(* Logix 5000 project; controller DC01 vendor 1 type 14 code 165 rev 32.12; software revision 32.04; part 12 of 13 *)
(* tags used below, declared in another part *)
   Always_Off : BOOL;
   Break_1stStation : BOOL;
   Break_LineWide : BOOL;
   Break_WorkCenter : BOOL;
   Break_Workstation : BOOL;
   FaultExists : CONTROL;
   LN04_MainLine_MSG : MESSAGE;
   Local_Timer : TIMER[30];
   ONS_0 : DINT;
   Scheduled_Units_Buffer : DINT;
   Shift_Reset : BOOL;
   Shift_Reset_ONS : BOOL;
   LN04_1st_Station_Break_Code : DINT;
   LN04_Additional_Break_Limit_Mins : DINT;
   LN04_BakeDrawer_MNT : DINT;
   LN04_Boxing_MNT : DINT;
   LN04_Console_MNT : DINT;
   LN04_Cooktop_MNT : DINT;
   LN04_Current_Shift_Duration_Mins : DINT;
   LN04_Current_Shift_Duration_wBreaks_Mins : DINT;
   LN04_DC_Controlled_Theoretical_Units : BOOL;
   LN04_Door_MNT : DINT;
   LN04_EStop_Funct_Test : DINT;
   LN04_EStop_Main_Panel : DINT;
   LN04_EStop_Main_Safety_Relay : DINT;
   LN04_EStop_MCC_Cabinet : DINT;
   LN04_FrontFrame_MNT : DINT;
   LN04_FunctionalTest_MNT : DINT;
   LN04_Ignition_NewSNModel : BOOL[32];
   LN04_Ignition_SNModelMSG : STRING[5];
   LN04_MachineOverAll_MNT : DINT;
   LN04_Main_Messages : DINT[250];
   LN04_MainBack_MNT : DINT;
   LN04_Messages_Barcode_SNModel : Barcode_SNModel;
   LN04_OT_Shift_Break_In_Minutes : DINT;
   LN04_OvenCavity_MNT : DINT;
   LN04_Pull_Cord_EStop_9111 : DINT;
   LN04_Pull_Cord_EStop_9112 : DINT;
   LN04_Pull_Cord_EStop_9200 : DINT;
   LN04_Pull_Cord_EStop_9201 : DINT;
   LN04_RackAndLiterature_MNT : DINT;
   LN04_Schedule : UDT_Current_Status;
   LN04_Schedule_Cycle_Timer : TIMER;
   LN04_Schedule_Max_Break_Duration : DINT;
   LN04_Schedule_Max_Break_Timer : TIMER;
   LN04_Schedule_TAKT : REAL;
   LN04_SidePanel_MNT : DINT;
   LN04_Standard_Shift_Break_In_Minutes : DINT;
   LN04_StorageDrawer_MNT : DINT;
   LN04_Theoretical_Units_Counter : COUNTER;
   LN04_Theoretical_Units_Counter_ONS : BOOL;
   LN04_Units_for_repair : DINT;
   LN04_Wiring_MNT : DINT;
   LN04EAM01 : DINT;
   LN04EAM02 : DINT;
   LN04ECM01 : DINT;
   LN04ECM02 : DINT;
   LN04EDM01 : DINT;
   LN04EEM01 : DINT;
   LN04EEM02 : DINT;
   LN04EEM03 : DINT;
   LN04EFM03 : DINT;
   LN04EGM01 : DINT;
   LN04EGM04 : DINT;
   LN04EGS01 : DINT;
   LN04EGS02 : DINT;
   LN04EGS03 : DINT;
   LN04EHM01 : DINT;
   LN04EHM02 : DINT;
   LN04EHM03 : DINT;
   LN04EHM04 : DINT;
   LN04EMM01 : DINT;
   LN04EMM03 : DINT;
   LN04NBS01 : DINT;
   LN04NBS02 : DINT;
   LN04NNM02 : DINT;
   LN04SAS01 : DINT;
   LN04SAS02 : DINT;
   LN04SDS01 : DINT;
   LN04SLS01 : DINT;
   LN04SLS02 : DINT;
   LN04SLS03 : DINT;
   LN04SNM02 : DINT;
   LN04WAM01 : DINT;
   LN04WBM01 : DINT;
   LN04WBM02 : DINT;
   LN04WCS01 : DINT;
   LN04WEM01 : DINT;
   LN04WEM02 : DINT;
   LN04WEM03 : DINT;
   LN04WFM01 : DINT;
   LN04WFM02 : DINT;
   LN04WFM03 : DINT;
   LN04WFM04 : DINT;
   LN04WFM05 : DINT;
   LN04WFS01 : DINT;
   LN04WFS02 : DINT;
   LN04WJM01 : DINT;
   LN04WJM02 : DINT;
   LN04WJM03 : DINT;
   LN04WKM01 : DINT;
   LN04WKM02 : DINT;
   LN04WKM03 : DINT;
   LN04WLM01 : DINT;
   LN04WMM01 : DINT;
   LN04WMM02 : DINT;
   LN04WMM03 : DINT;
   LN04WMM04 : DINT;
   LN04WNM01 : DINT;
(* LN04, continued *)

ROUTINE R02_CurrentShift_Calcs   (* ladder *)
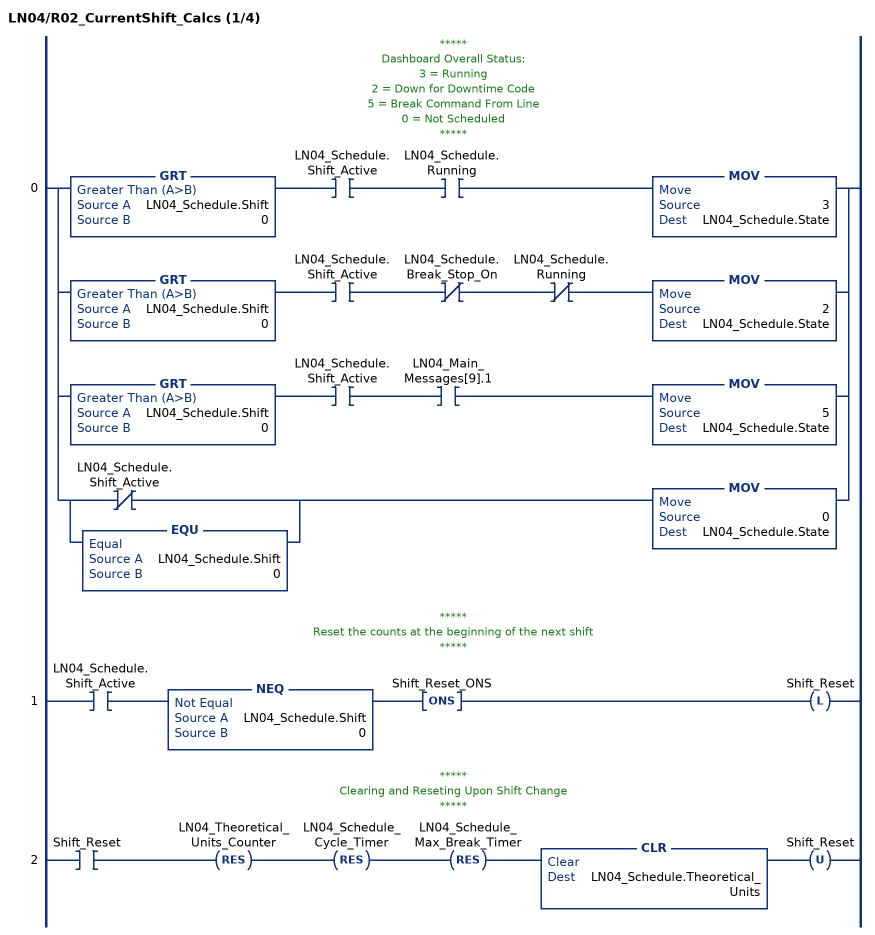
   // *****
   // Dashboard Overall Status:
   // 3 = Running
   // 2 = Down for Downtime Code
   // 5 = Break Command From Line
   // 0 = Not Scheduled
   // *****
   0: [GRT(LN04_Schedule.Shift,0) XIC(LN04_Schedule.Shift_Active) XIC(LN04_Schedule.Running) MOV(3,LN04_Schedule.State) ,GRT(LN04_Schedule.Shift,0) XIC(LN04_Schedule.Shift_Active) XIO(LN04_Schedule.Break_Stop_On) XIO(LN04_Schedule.Running) MOV(2,LN04_Schedule.State) ,GRT(LN04_Schedule.Shift,0) XIC(LN04_Schedule.Shift_Active) XIC(LN04_Main_Messages[9].1) MOV(5,LN04_Schedule.State) ,[XIO(LN04_Schedule.Shift_Active) ,EQU(LN04_Schedule.Shift,0) ] MOV(0,LN04_Schedule.State) ];
   // *****
   // Reset the counts at the beginning of the next shift
   // *****
   1: XIC(LN04_Schedule.Shift_Active)NEQ(LN04_Schedule.Shift,0)ONS(Shift_Reset_ONS)OTL(Shift_Reset);
   // *****
   // Clearing and Reseting Upon Shift Change
   // *****
   2: XIC(Shift_Reset)RES(LN04_Theoretical_Units_Counter)RES(LN04_Schedule_Cycle_Timer)RES(LN04_Schedule_Max_Break_Timer)CLR(LN04_Schedule.Theoretical_Units)OTU(Shift_Reset);
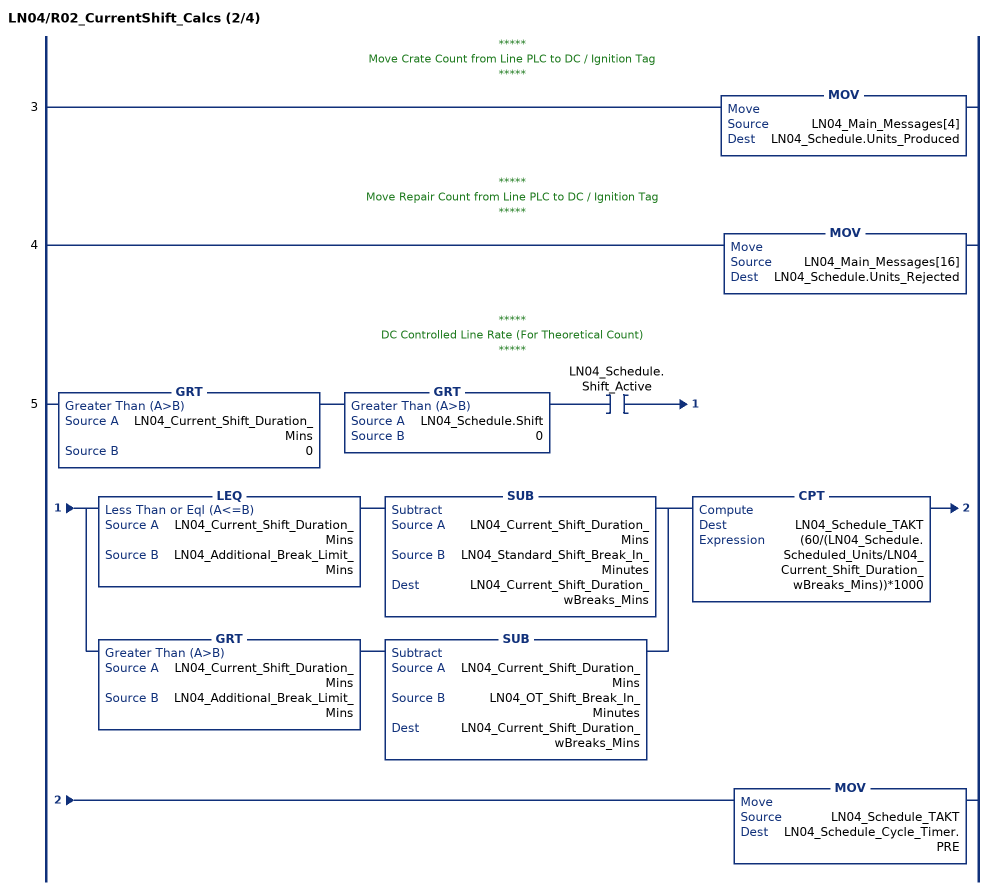
   // *****
   // Move Crate Count from Line PLC to DC / Ignition Tag
   // *****
   3: MOV(LN04_Main_Messages[4],LN04_Schedule.Units_Produced);
   // *****
   // Move Repair Count from Line PLC to DC / Ignition Tag
   // *****
   4: MOV(LN04_Main_Messages[16],LN04_Schedule.Units_Rejected);
   // *****
   // DC Controlled Line Rate (For Theoretical Count)
   // *****
   5: GRT(LN04_Current_Shift_Duration_Mins,0)GRT(LN04_Schedule.Shift,0)XIC(LN04_Schedule.Shift_Active)[LEQ(LN04_Current_Shift_Duration_Mins,LN04_Additional_Break_Limit_Mins) SUB(LN04_Current_Shift_Duration_Mins,LN04_Standard_Shift_Break_In_Minutes,LN04_Current_Shift_Duration_wBreaks_Mins) ,GRT(LN04_Current_Shift_Duration_Mins,LN04_Additional_Break_Limit_Mins) SUB(LN04_Current_Shift_Duration_Mins,LN04_OT_Shift_Break_In_Minutes,LN04_Current_Shift_Duration_wBreaks_Mins) ]CPT(LN04_Schedule_TAKT,(60/(LN04_Schedule.Scheduled_Units/LN04_Current_Shift_Duration_wBreaks_Mins))*1000)MOV(LN04_Schedule_TAKT,LN04_Schedule_Cycle_Timer.PRE);
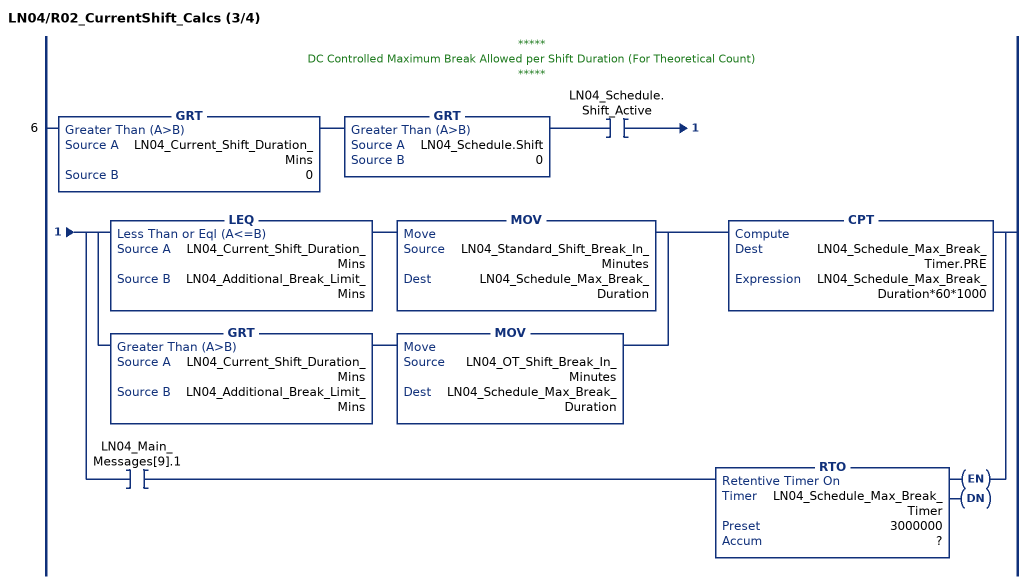
   // *****
   // DC Controlled Maximum Break Allowed per Shift Duration (For Theoretical Count)
   // *****
   6: GRT(LN04_Current_Shift_Duration_Mins,0)GRT(LN04_Schedule.Shift,0)XIC(LN04_Schedule.Shift_Active)[[LEQ(LN04_Current_Shift_Duration_Mins,LN04_Additional_Break_Limit_Mins) MOV(LN04_Standard_Shift_Break_In_Minutes,LN04_Schedule_Max_Break_Duration) ,GRT(LN04_Current_Shift_Duration_Mins,LN04_Additional_Break_Limit_Mins) MOV(LN04_OT_Shift_Break_In_Minutes,LN04_Schedule_Max_Break_Duration) ] CPT(LN04_Schedule_Max_Break_Timer.PRE,LN04_Schedule_Max_Break_Duration*60*1000) ,XIC(LN04_Main_Messages[9].1) RTO(LN04_Schedule_Max_Break_Timer,?,?) ];
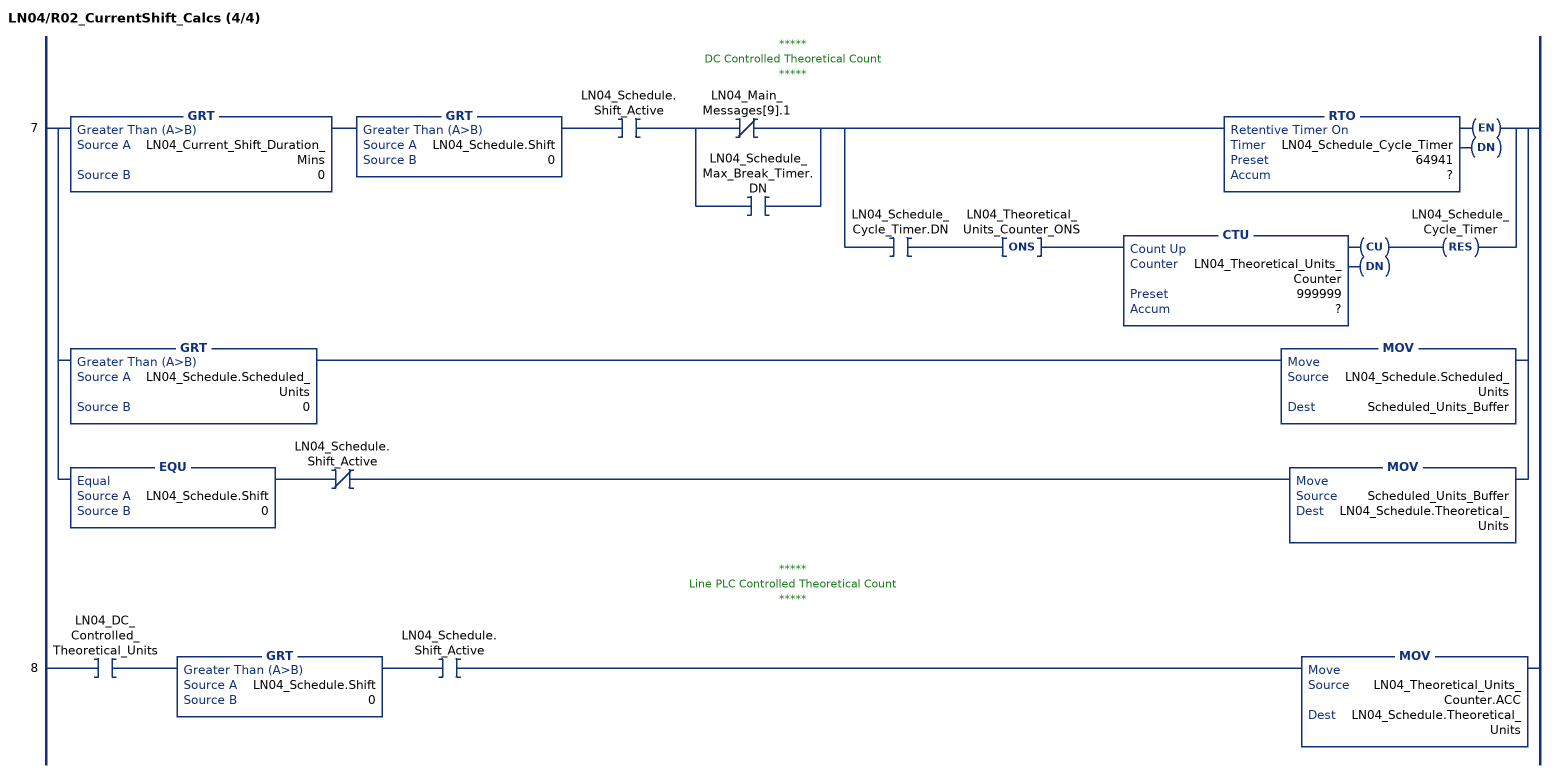
   // *****
   // DC Controlled Theoretical Count
   // *****
   7: [GRT(LN04_Current_Shift_Duration_Mins,0) GRT(LN04_Schedule.Shift,0) XIC(LN04_Schedule.Shift_Active) [XIO(LN04_Main_Messages[9].1) ,XIC(LN04_Schedule_Max_Break_Timer.DN) ] [RTO(LN04_Schedule_Cycle_Timer,?,?) ,XIC(LN04_Schedule_Cycle_Timer.DN) ONS(LN04_Theoretical_Units_Counter_ONS) CTU(LN04_Theoretical_Units_Counter,?,?) RES(LN04_Schedule_Cycle_Timer) ] ,GRT(LN04_Schedule.Scheduled_Units,0) MOV(LN04_Schedule.Scheduled_Units,Scheduled_Units_Buffer) ,EQU(LN04_Schedule.Shift,0) XIO(LN04_Schedule.Shift_Active) MOV(Scheduled_Units_Buffer,LN04_Schedule.Theoretical_Units) ];
   // *****
   // Line PLC Controlled Theoretical Count
   // *****
   8: XIC(LN04_DC_Controlled_Theoretical_Units)GRT(LN04_Schedule.Shift,0)XIC(LN04_Schedule.Shift_Active)MOV(LN04_Theoretical_Units_Counter.ACC,LN04_Schedule.Theoretical_Units);
END_ROUTINE

ROUTINE R03_DataFromLines   (* ladder *)
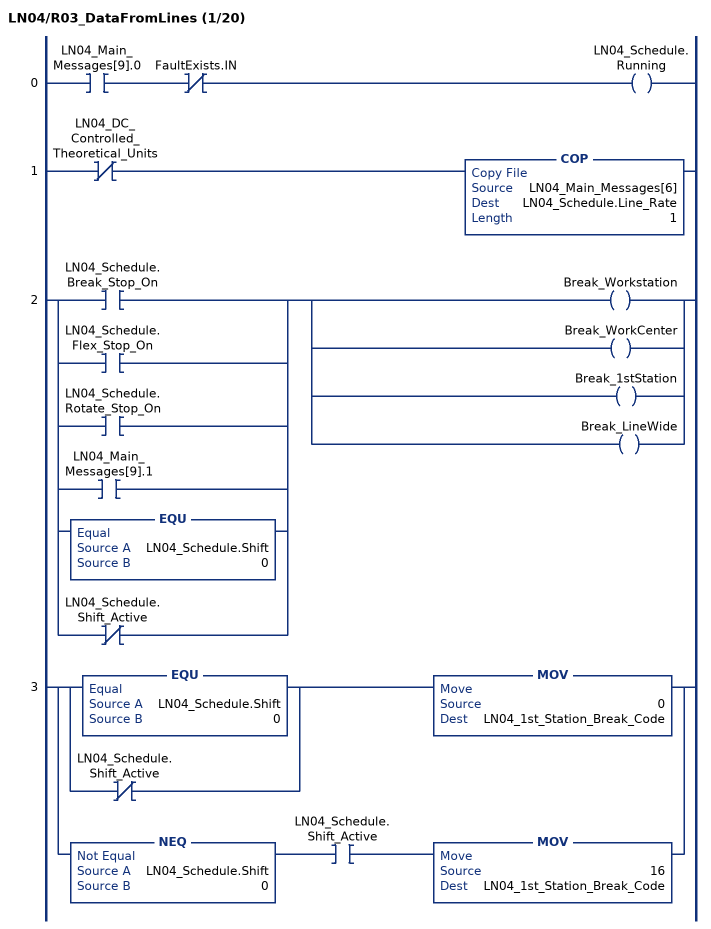
   0: XIC(LN04_Main_Messages[9].0)XIO(FaultExists.IN)OTE(LN04_Schedule.Running);
   1: XIO(LN04_DC_Controlled_Theoretical_Units)COP(LN04_Main_Messages[6],LN04_Schedule.Line_Rate,1);
   2: [XIC(LN04_Schedule.Break_Stop_On) ,XIC(LN04_Schedule.Flex_Stop_On) ,XIC(LN04_Schedule.Rotate_Stop_On) ,XIC(LN04_Main_Messages[9].1) ,EQU(LN04_Schedule.Shift,0) ,XIO(LN04_Schedule.Shift_Active) ][OTE(Break_Workstation) ,OTE(Break_WorkCenter) ,OTE(Break_1stStation) ,OTE(Break_LineWide) ];
   3: [[EQU(LN04_Schedule.Shift,0) ,XIO(LN04_Schedule.Shift_Active) ] MOV(0,LN04_1st_Station_Break_Code) ,NEQ(LN04_Schedule.Shift,0) XIC(LN04_Schedule.Shift_Active) MOV(16,LN04_1st_Station_Break_Code) ];
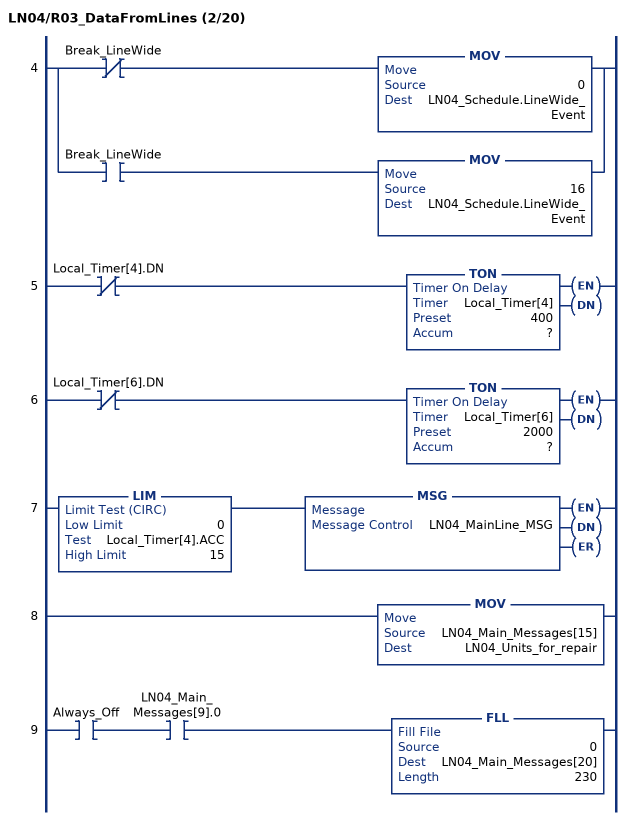
   4: [XIO(Break_LineWide) MOV(0,LN04_Schedule.LineWide_Event) ,XIC(Break_LineWide) MOV(16,LN04_Schedule.LineWide_Event) ];
   5: XIO(Local_Timer[4].DN)TON(Local_Timer[4],?,?);
   6: XIO(Local_Timer[6].DN)TON(Local_Timer[6],?,?);
   7: LIM(0,Local_Timer[4].ACC,15)MSG(LN04_MainLine_MSG);
   8: MOV(LN04_Main_Messages[15],LN04_Units_for_repair);
   9: XIC(Always_Off)XIC(LN04_Main_Messages[9].0)FLL(0,LN04_Main_Messages[20],230);
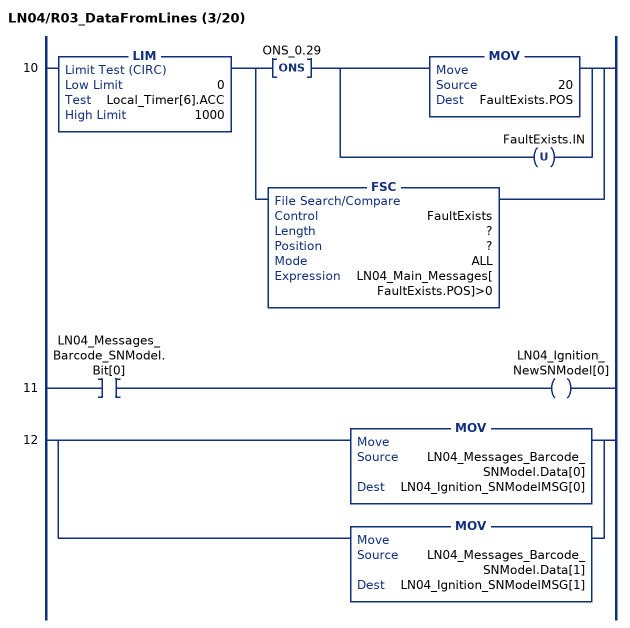
   10: LIM(0,Local_Timer[6].ACC,1000)[ONS(ONS_0.29) [MOV(20,FaultExists.POS) ,OTU(FaultExists.IN) ] ,FSC(FaultExists,?,?,ALL,LN04_Main_Messages[FaultExists.POS]>0) ];
   11: XIC(LN04_Messages_Barcode_SNModel.Bit[0])OTE(LN04_Ignition_NewSNModel[0]);
   12: [MOV(LN04_Messages_Barcode_SNModel.Data[0],LN04_Ignition_SNModelMSG[0]) ,MOV(LN04_Messages_Barcode_SNModel.Data[1],LN04_Ignition_SNModelMSG[1]) ];
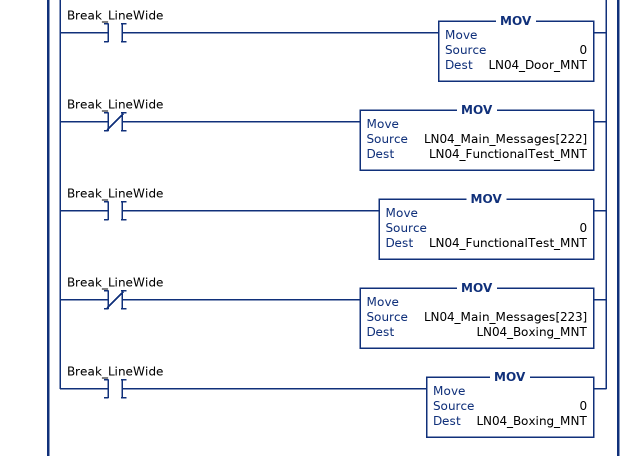
   13: [XIO(Break_LineWide) MOV(LN04_Main_Messages[20],LN04_MachineOverAll_MNT) ,XIC(Break_LineWide) MOV(0,LN04_MachineOverAll_MNT) ,XIO(Break_LineWide) MOV(LN04_Main_Messages[21],LN04_FrontFrame_MNT) ,XIC(Break_LineWide) MOV(0,LN04_FrontFrame_MNT) ,XIO(Break_LineWide) MOV(LN04_Main_Messages[22],LN04_OvenCavity_MNT) ,XIC(Break_LineWide) MOV(0,LN04_OvenCavity_MNT) ,XIO(Break_LineWide) MOV(LN04_Main_Messages[23],LN04_BakeDrawer_MNT) ,XIC(Break_LineWide) MOV(0,LN04_BakeDrawer_MNT) ,XIO(Break_LineWide) MOV(LN04_Main_Messages[24],LN04_MainBack_MNT) ,XIC(Break_LineWide) MOV(0,LN04_MainBack_MNT) ,XIO(Break_LineWide) MOV(LN04_Main_Messages[25],LN04_SidePanel_MNT) ,XIC(Break_LineWide) MOV(0,LN04_SidePanel_MNT) ,XIO(Break_LineWide) MOV(LN04_Main_Messages[26],LN04_Cooktop_MNT) ,XIC(Break_LineWide) MOV(0,LN04_Cooktop_MNT) ,XIO(Break_LineWide) MOV(LN04_Main_Messages[27],LN04_Console_MNT) ,XIC(Break_LineWide) MOV(0,LN04_Console_MNT) ,XIO(Break_LineWide) MOV(LN04_Main_Messages[28],LN04_Wiring_MNT) ,XIC(Break_LineWide) MOV(0,LN04_Wiring_MNT) ,XIO(Break_LineWide) MOV(LN04_Main_Messages[29],LN04_StorageDrawer_MNT) ,XIC(Break_LineWide) MOV(0,LN04_StorageDrawer_MNT) ,XIO(Break_LineWide) MOV(LN04_Main_Messages[220],LN04_RackAndLiterature_MNT) ,XIC(Break_LineWide) MOV(0,LN04_RackAndLiterature_MNT) ,XIO(Break_LineWide) MOV(LN04_Main_Messages[221],LN04_Door_MNT) ,XIC(Break_LineWide) MOV(0,LN04_Door_MNT) ,XIO(Break_LineWide) MOV(LN04_Main_Messages[222],LN04_FunctionalTest_MNT) ,XIC(Break_LineWide) MOV(0,LN04_FunctionalTest_MNT) ,XIO(Break_LineWide) MOV(LN04_Main_Messages[223],LN04_Boxing_MNT) ,XIC(Break_LineWide) MOV(0,LN04_Boxing_MNT) ];
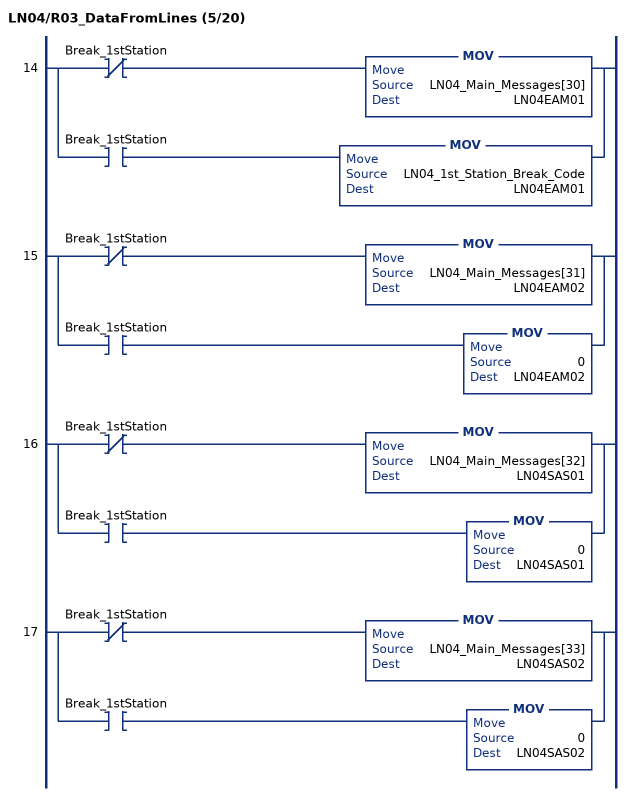
   14: [XIO(Break_1stStation) MOV(LN04_Main_Messages[30],LN04EAM01) ,XIC(Break_1stStation) MOV(LN04_1st_Station_Break_Code,LN04EAM01) ];
   15: [XIO(Break_1stStation) MOV(LN04_Main_Messages[31],LN04EAM02) ,XIC(Break_1stStation) MOV(0,LN04EAM02) ];
   16: [XIO(Break_1stStation) MOV(LN04_Main_Messages[32],LN04SAS01) ,XIC(Break_1stStation) MOV(0,LN04SAS01) ];
   17: [XIO(Break_1stStation) MOV(LN04_Main_Messages[33],LN04SAS02) ,XIC(Break_1stStation) MOV(0,LN04SAS02) ];
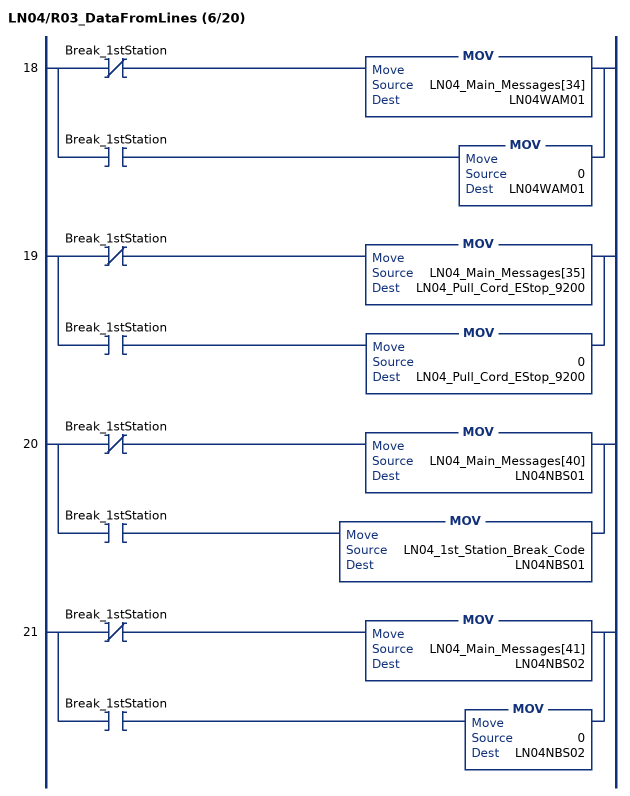
   18: [XIO(Break_1stStation) MOV(LN04_Main_Messages[34],LN04WAM01) ,XIC(Break_1stStation) MOV(0,LN04WAM01) ];
   19: [XIO(Break_1stStation) MOV(LN04_Main_Messages[35],LN04_Pull_Cord_EStop_9200) ,XIC(Break_1stStation) MOV(0,LN04_Pull_Cord_EStop_9200) ];
   20: [XIO(Break_1stStation) MOV(LN04_Main_Messages[40],LN04NBS01) ,XIC(Break_1stStation) MOV(LN04_1st_Station_Break_Code,LN04NBS01) ];
   21: [XIO(Break_1stStation) MOV(LN04_Main_Messages[41],LN04NBS02) ,XIC(Break_1stStation) MOV(0,LN04NBS02) ];
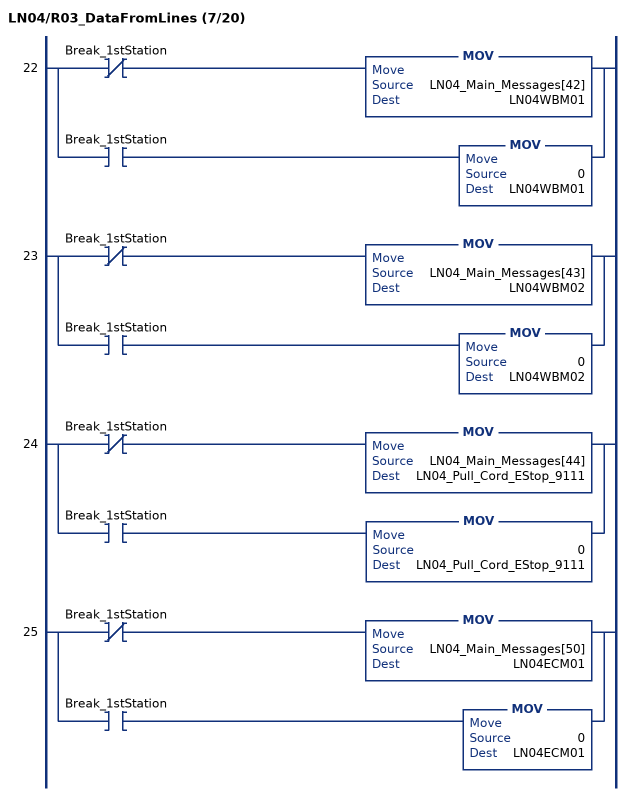
   22: [XIO(Break_1stStation) MOV(LN04_Main_Messages[42],LN04WBM01) ,XIC(Break_1stStation) MOV(0,LN04WBM01) ];
   23: [XIO(Break_1stStation) MOV(LN04_Main_Messages[43],LN04WBM02) ,XIC(Break_1stStation) MOV(0,LN04WBM02) ];
   24: [XIO(Break_1stStation) MOV(LN04_Main_Messages[44],LN04_Pull_Cord_EStop_9111) ,XIC(Break_1stStation) MOV(0,LN04_Pull_Cord_EStop_9111) ];
   25: [XIO(Break_1stStation) MOV(LN04_Main_Messages[50],LN04ECM01) ,XIC(Break_1stStation) MOV(0,LN04ECM01) ];
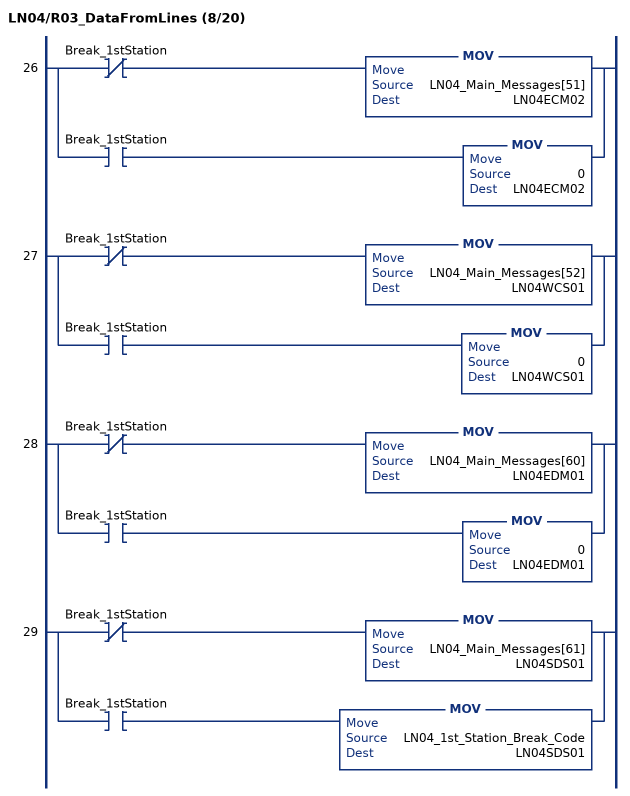
   26: [XIO(Break_1stStation) MOV(LN04_Main_Messages[51],LN04ECM02) ,XIC(Break_1stStation) MOV(0,LN04ECM02) ];
   27: [XIO(Break_1stStation) MOV(LN04_Main_Messages[52],LN04WCS01) ,XIC(Break_1stStation) MOV(0,LN04WCS01) ];
   28: [XIO(Break_1stStation) MOV(LN04_Main_Messages[60],LN04EDM01) ,XIC(Break_1stStation) MOV(0,LN04EDM01) ];
   29: [XIO(Break_1stStation) MOV(LN04_Main_Messages[61],LN04SDS01) ,XIC(Break_1stStation) MOV(LN04_1st_Station_Break_Code,LN04SDS01) ];
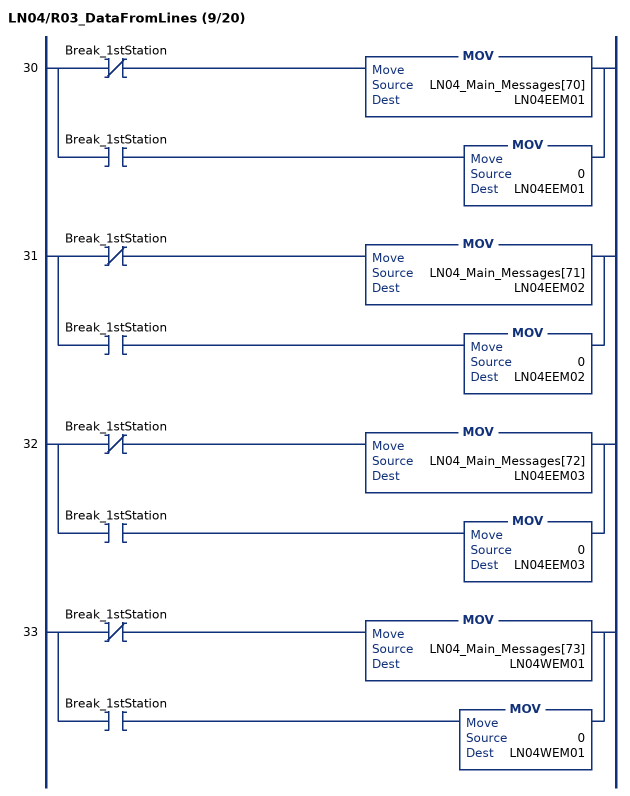
   30: [XIO(Break_1stStation) MOV(LN04_Main_Messages[70],LN04EEM01) ,XIC(Break_1stStation) MOV(0,LN04EEM01) ];
   31: [XIO(Break_1stStation) MOV(LN04_Main_Messages[71],LN04EEM02) ,XIC(Break_1stStation) MOV(0,LN04EEM02) ];
   32: [XIO(Break_1stStation) MOV(LN04_Main_Messages[72],LN04EEM03) ,XIC(Break_1stStation) MOV(0,LN04EEM03) ];
   33: [XIO(Break_1stStation) MOV(LN04_Main_Messages[73],LN04WEM01) ,XIC(Break_1stStation) MOV(0,LN04WEM01) ];
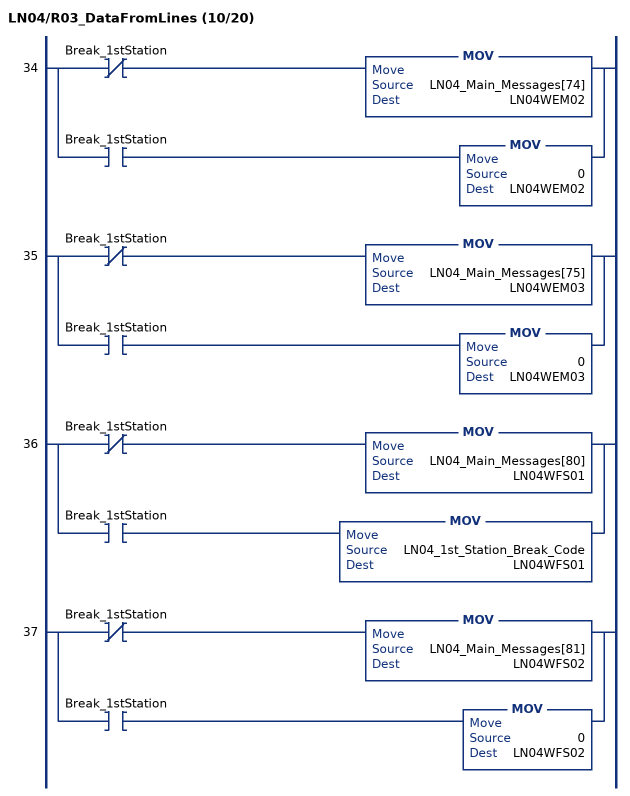
   34: [XIO(Break_1stStation) MOV(LN04_Main_Messages[74],LN04WEM02) ,XIC(Break_1stStation) MOV(0,LN04WEM02) ];
   35: [XIO(Break_1stStation) MOV(LN04_Main_Messages[75],LN04WEM03) ,XIC(Break_1stStation) MOV(0,LN04WEM03) ];
   36: [XIO(Break_1stStation) MOV(LN04_Main_Messages[80],LN04WFS01) ,XIC(Break_1stStation) MOV(LN04_1st_Station_Break_Code,LN04WFS01) ];
   37: [XIO(Break_1stStation) MOV(LN04_Main_Messages[81],LN04WFS02) ,XIC(Break_1stStation) MOV(0,LN04WFS02) ];
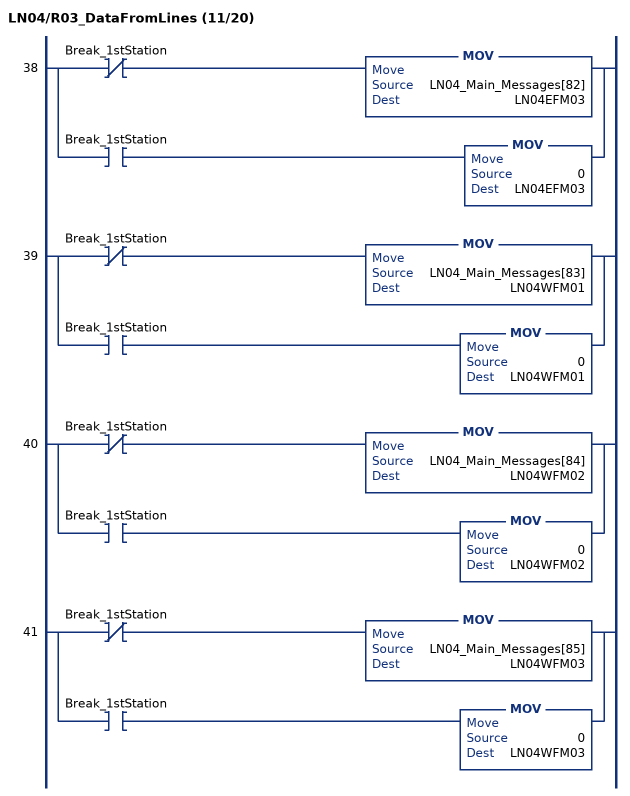
   38: [XIO(Break_1stStation) MOV(LN04_Main_Messages[82],LN04EFM03) ,XIC(Break_1stStation) MOV(0,LN04EFM03) ];
   39: [XIO(Break_1stStation) MOV(LN04_Main_Messages[83],LN04WFM01) ,XIC(Break_1stStation) MOV(0,LN04WFM01) ];
   40: [XIO(Break_1stStation) MOV(LN04_Main_Messages[84],LN04WFM02) ,XIC(Break_1stStation) MOV(0,LN04WFM02) ];
   41: [XIO(Break_1stStation) MOV(LN04_Main_Messages[85],LN04WFM03) ,XIC(Break_1stStation) MOV(0,LN04WFM03) ];
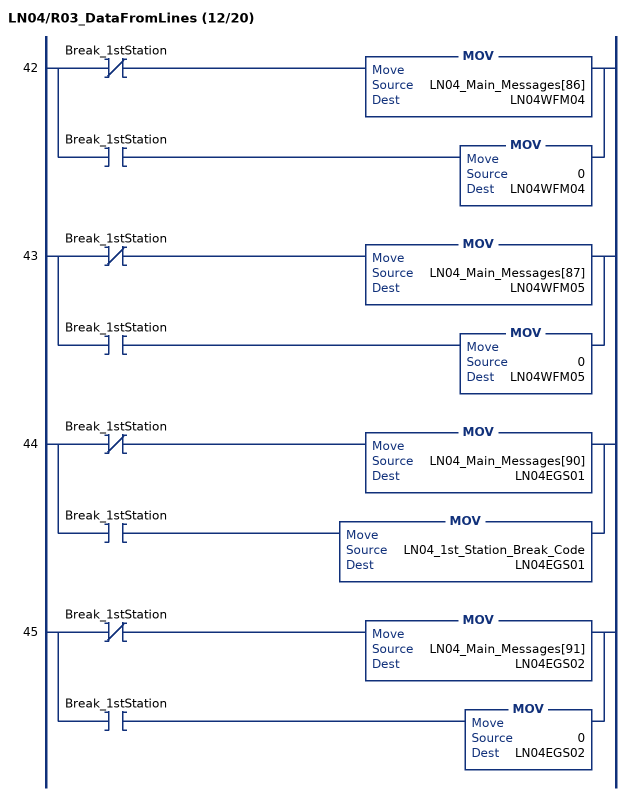
   42: [XIO(Break_1stStation) MOV(LN04_Main_Messages[86],LN04WFM04) ,XIC(Break_1stStation) MOV(0,LN04WFM04) ];
   43: [XIO(Break_1stStation) MOV(LN04_Main_Messages[87],LN04WFM05) ,XIC(Break_1stStation) MOV(0,LN04WFM05) ];
   44: [XIO(Break_1stStation) MOV(LN04_Main_Messages[90],LN04EGS01) ,XIC(Break_1stStation) MOV(LN04_1st_Station_Break_Code,LN04EGS01) ];
   45: [XIO(Break_1stStation) MOV(LN04_Main_Messages[91],LN04EGS02) ,XIC(Break_1stStation) MOV(0,LN04EGS02) ];
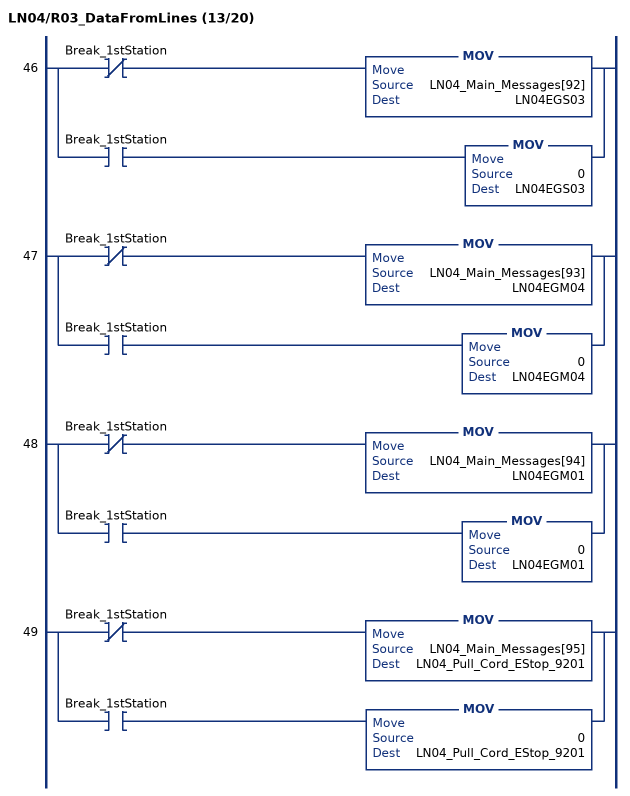
   46: [XIO(Break_1stStation) MOV(LN04_Main_Messages[92],LN04EGS03) ,XIC(Break_1stStation) MOV(0,LN04EGS03) ];
   47: [XIO(Break_1stStation) MOV(LN04_Main_Messages[93],LN04EGM04) ,XIC(Break_1stStation) MOV(0,LN04EGM04) ];
   48: [XIO(Break_1stStation) MOV(LN04_Main_Messages[94],LN04EGM01) ,XIC(Break_1stStation) MOV(0,LN04EGM01) ];
   49: [XIO(Break_1stStation) MOV(LN04_Main_Messages[95],LN04_Pull_Cord_EStop_9201) ,XIC(Break_1stStation) MOV(0,LN04_Pull_Cord_EStop_9201) ];
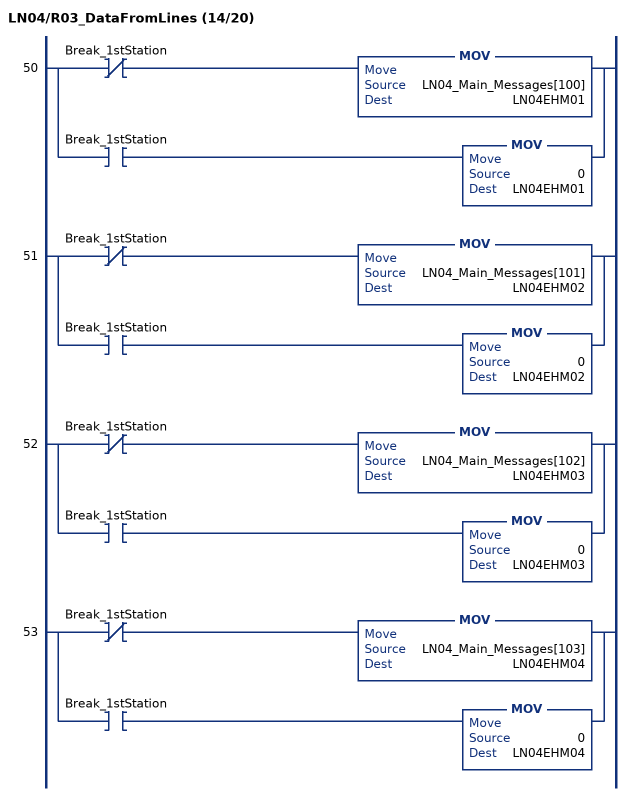
   50: [XIO(Break_1stStation) MOV(LN04_Main_Messages[100],LN04EHM01) ,XIC(Break_1stStation) MOV(0,LN04EHM01) ];
   51: [XIO(Break_1stStation) MOV(LN04_Main_Messages[101],LN04EHM02) ,XIC(Break_1stStation) MOV(0,LN04EHM02) ];
   52: [XIO(Break_1stStation) MOV(LN04_Main_Messages[102],LN04EHM03) ,XIC(Break_1stStation) MOV(0,LN04EHM03) ];
   53: [XIO(Break_1stStation) MOV(LN04_Main_Messages[103],LN04EHM04) ,XIC(Break_1stStation) MOV(0,LN04EHM04) ];
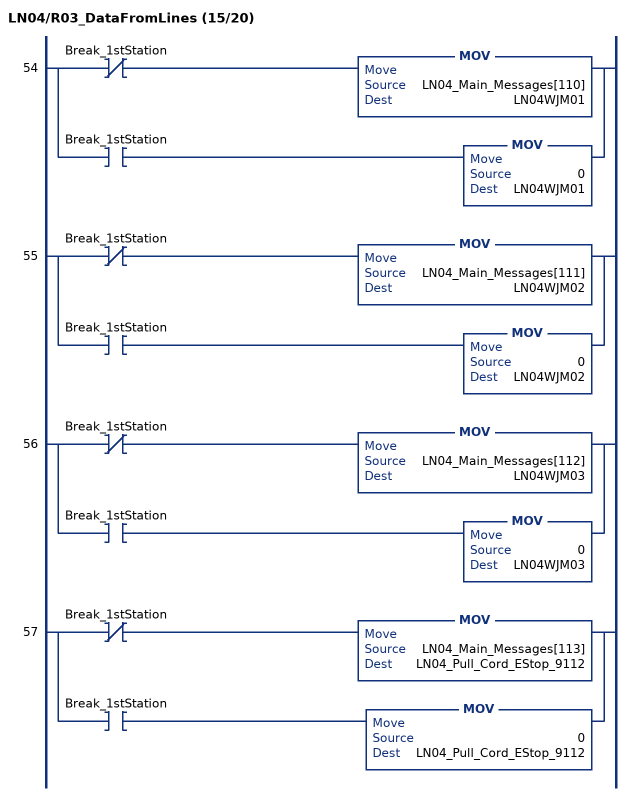
   54: [XIO(Break_1stStation) MOV(LN04_Main_Messages[110],LN04WJM01) ,XIC(Break_1stStation) MOV(0,LN04WJM01) ];
   55: [XIO(Break_1stStation) MOV(LN04_Main_Messages[111],LN04WJM02) ,XIC(Break_1stStation) MOV(0,LN04WJM02) ];
   56: [XIO(Break_1stStation) MOV(LN04_Main_Messages[112],LN04WJM03) ,XIC(Break_1stStation) MOV(0,LN04WJM03) ];
   57: [XIO(Break_1stStation) MOV(LN04_Main_Messages[113],LN04_Pull_Cord_EStop_9112) ,XIC(Break_1stStation) MOV(0,LN04_Pull_Cord_EStop_9112) ];
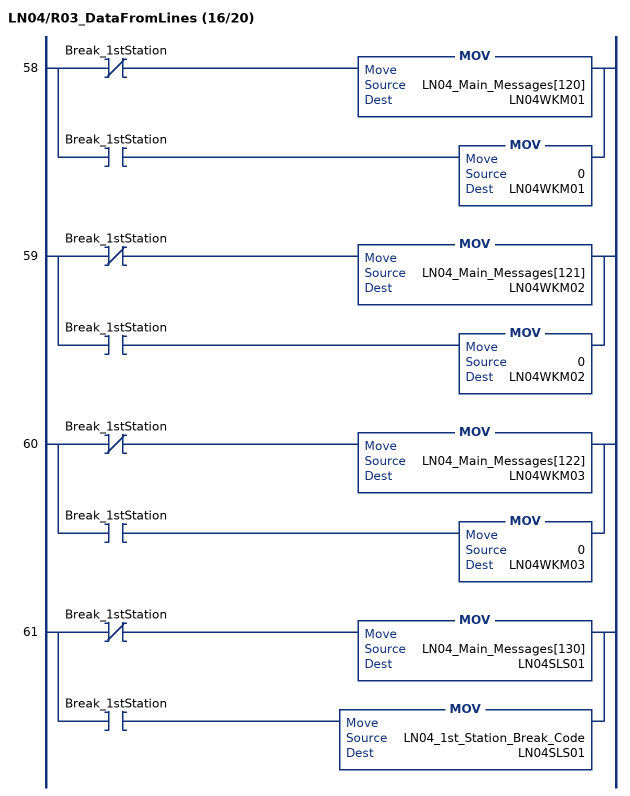
   58: [XIO(Break_1stStation) MOV(LN04_Main_Messages[120],LN04WKM01) ,XIC(Break_1stStation) MOV(0,LN04WKM01) ];
   59: [XIO(Break_1stStation) MOV(LN04_Main_Messages[121],LN04WKM02) ,XIC(Break_1stStation) MOV(0,LN04WKM02) ];
   60: [XIO(Break_1stStation) MOV(LN04_Main_Messages[122],LN04WKM03) ,XIC(Break_1stStation) MOV(0,LN04WKM03) ];
   61: [XIO(Break_1stStation) MOV(LN04_Main_Messages[130],LN04SLS01) ,XIC(Break_1stStation) MOV(LN04_1st_Station_Break_Code,LN04SLS01) ];
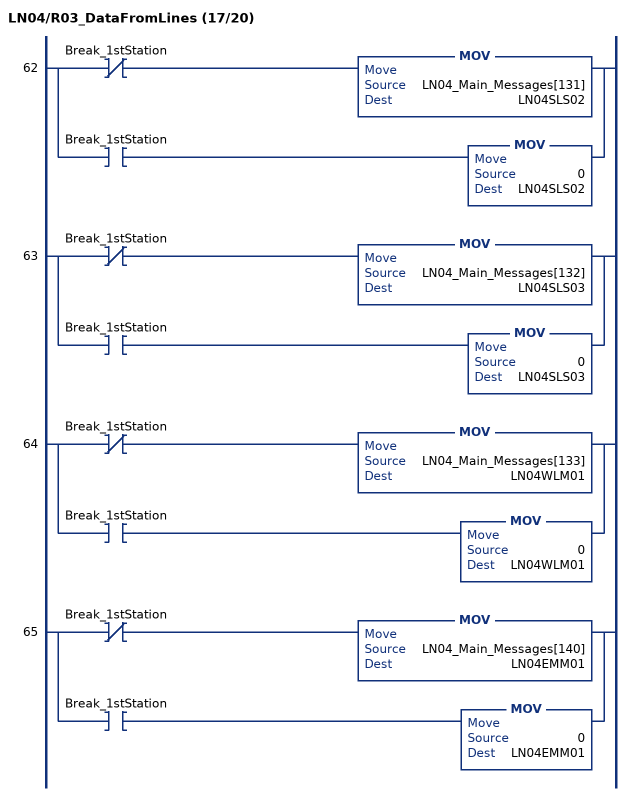
   62: [XIO(Break_1stStation) MOV(LN04_Main_Messages[131],LN04SLS02) ,XIC(Break_1stStation) MOV(0,LN04SLS02) ];
   63: [XIO(Break_1stStation) MOV(LN04_Main_Messages[132],LN04SLS03) ,XIC(Break_1stStation) MOV(0,LN04SLS03) ];
   64: [XIO(Break_1stStation) MOV(LN04_Main_Messages[133],LN04WLM01) ,XIC(Break_1stStation) MOV(0,LN04WLM01) ];
   65: [XIO(Break_1stStation) MOV(LN04_Main_Messages[140],LN04EMM01) ,XIC(Break_1stStation) MOV(0,LN04EMM01) ];
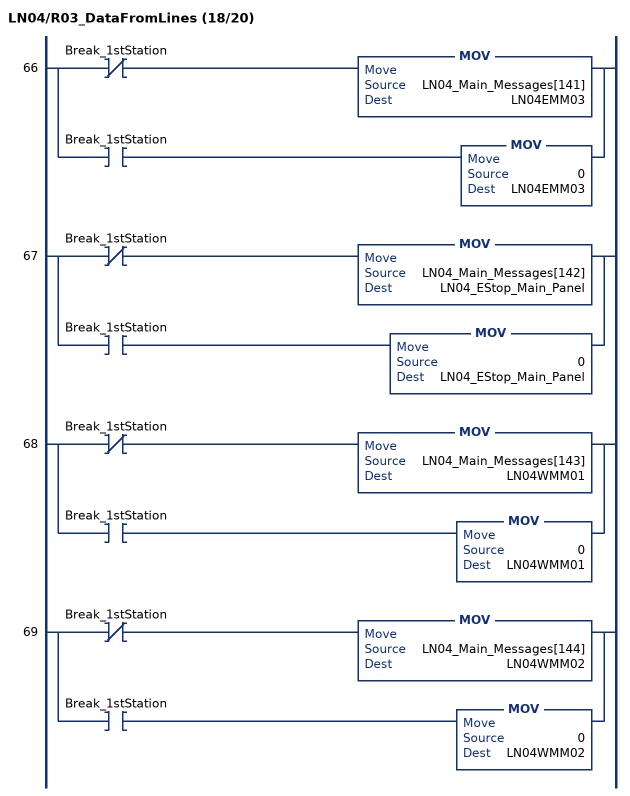
   66: [XIO(Break_1stStation) MOV(LN04_Main_Messages[141],LN04EMM03) ,XIC(Break_1stStation) MOV(0,LN04EMM03) ];
   67: [XIO(Break_1stStation) MOV(LN04_Main_Messages[142],LN04_EStop_Main_Panel) ,XIC(Break_1stStation) MOV(0,LN04_EStop_Main_Panel) ];
   68: [XIO(Break_1stStation) MOV(LN04_Main_Messages[143],LN04WMM01) ,XIC(Break_1stStation) MOV(0,LN04WMM01) ];
   69: [XIO(Break_1stStation) MOV(LN04_Main_Messages[144],LN04WMM02) ,XIC(Break_1stStation) MOV(0,LN04WMM02) ];
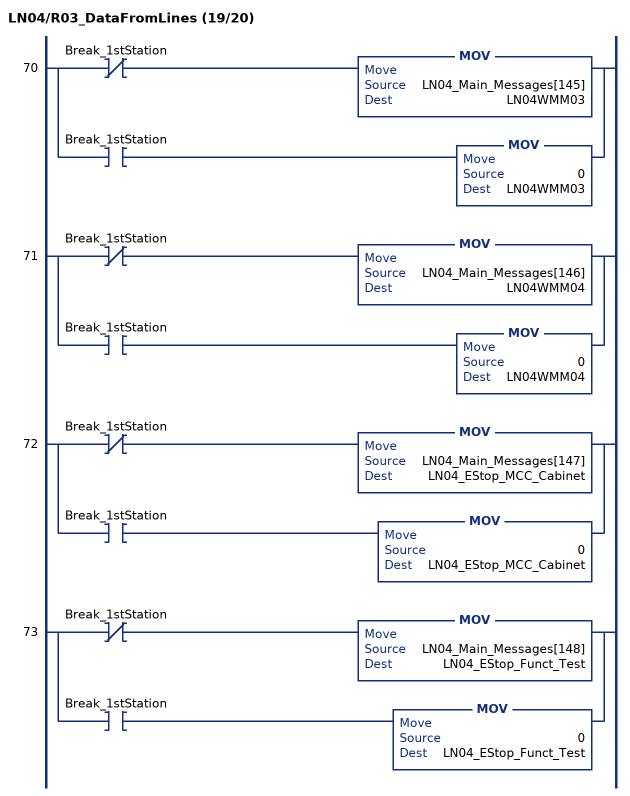
   70: [XIO(Break_1stStation) MOV(LN04_Main_Messages[145],LN04WMM03) ,XIC(Break_1stStation) MOV(0,LN04WMM03) ];
   71: [XIO(Break_1stStation) MOV(LN04_Main_Messages[146],LN04WMM04) ,XIC(Break_1stStation) MOV(0,LN04WMM04) ];
   72: [XIO(Break_1stStation) MOV(LN04_Main_Messages[147],LN04_EStop_MCC_Cabinet) ,XIC(Break_1stStation) MOV(0,LN04_EStop_MCC_Cabinet) ];
   73: [XIO(Break_1stStation) MOV(LN04_Main_Messages[148],LN04_EStop_Funct_Test) ,XIC(Break_1stStation) MOV(0,LN04_EStop_Funct_Test) ];
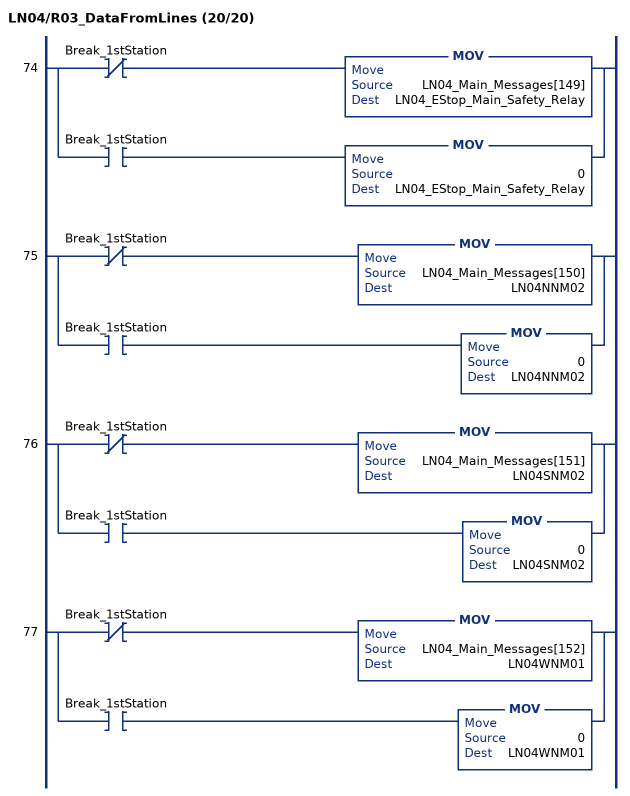
   74: [XIO(Break_1stStation) MOV(LN04_Main_Messages[149],LN04_EStop_Main_Safety_Relay) ,XIC(Break_1stStation) MOV(0,LN04_EStop_Main_Safety_Relay) ];
   75: [XIO(Break_1stStation) MOV(LN04_Main_Messages[150],LN04NNM02) ,XIC(Break_1stStation) MOV(0,LN04NNM02) ];
   76: [XIO(Break_1stStation) MOV(LN04_Main_Messages[151],LN04SNM02) ,XIC(Break_1stStation) MOV(0,LN04SNM02) ];
   77: [XIO(Break_1stStation) MOV(LN04_Main_Messages[152],LN04WNM01) ,XIC(Break_1stStation) MOV(0,LN04WNM01) ];
END_ROUTINE
